PROGRAM MAIN
VAR
	bBadPartDetected: BOOL := FALSE;
	bRejectArmEnabled: BOOL := FALSE;
	tTravelTimer: TON;
	tPushTimer: TON;
	bRejectMemory: BOOL := FALSE;
	
END_VAR

IF bBadPartDetected THEN
	bRejectMemory := TRUE;
END_IF;
tTravelTimer(IN:= bRejectMemory, PT := T#3S);
tPushTimer(IN:= tTravelTimer.Q, PT:= T#1S);
IF NOT tPushTimer.Q AND bRejectMemory AND tTravelTimer.Q THEN
	bRejectArmEnabled := TRUE;
ELSE;
	bRejectArmEnabled := FALSE;
END_IF;
IF tPushTimer.Q AND tTravelTimer.Q THEN
	bBadPartDetected := FALSE;
	bRejectMemory := FALSE;
END_IF;

END_PROGRAM

(* stored: Version 1.1.0.1, ProductVersion 3.1.4024.16
   POU MAIN: Id {d81b1351-9aef-4f54-aa3e-f196943c2498}, SpecialFunc None *)
